FUNCTION_BLOCK E_SPLIT
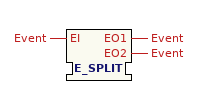
  EVENT_INPUT
    EI;
  END_EVENT
  EVENT_OUTPUT
    EO1;
    EO2;
  END_EVENT
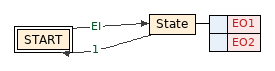
  EC_STATES
    START;
    State : -> EO1, -> EO2;
  END_STATES
  EC_TRANSITIONS
    START TO State := EI;
    State TO START := 1;
  END_TRANSITIONS
END_FUNCTION_BLOCK
